/// Implicitly generated code : DO NOT EDIT!!!
/// CheckBounds is used to check for range overflows
{attribute 'check_bounds' := ''}
{attribute 'no_check' := ''}
FUNCTION CheckBounds : DINT
VAR_INPUT
	index: DINT;
	lower: DINT;
	upper: DINT;
END_VAR

// align bounds 
CheckBounds := MIN(upper, MAX(lower, index));

// if index changed, report error
IF CheckBounds <> index THEN
	GVL_Supervision.aCodeErr[eCodeError_bounds] := TRUE;
END_IF

END_FUNCTION

(* stored: Version 1.1.0.1, ProductVersion 3.1.4022.9
   POU CheckBounds: Id {78c83943-6d9c-4d3b-944d-42aa3c0016a6}, SpecialFunc None *)
